INTERFACE I_Serializer

METHOD Serialize : HRESULT
VAR_INPUT
	anyArg	: ANY;
END_VAR
VAR_IN_OUT
	sJsonDocument	: T_VerifyContent;
END_VAR
END_METHOD

END_INTERFACE

(* stored: Version 1.1.0.1, ProductVersion 3.1.4026.18
   Itf I_Serializer: Id {73355309-3f85-459c-acba-6d5c99a77725}
   Method Serialize: Id {54315dda-706c-44e0-b44e-f8f81fc5f914} *)
